FUNCTION_BLOCK FB_count
VAR_INPUT
	Add_Time:TIME;
END_VAR
VAR_OUTPUT
	count:INT;
END_VAR
VAR
	ton1:TON;
	a:INT;
END_VAR

ton1(IN:=NOT ton1.Q  , PT:=Add_Time , Q=> , ET=> );
IF ton1.Q THEN 
	count:=count+1;
END_IF
IF count>=1000 THEN 
	count:=0;
END_IF

END_FUNCTION_BLOCK

(* stored: Version 1.1.0.1, ProductVersion 3.1.4024.11
   POU FB_count: Id {7b951bcc-d3ad-48a1-aea4-f34a926b184d}, SpecialFunc None *)
